# EPICS autosave request: iocBoot/ioc32IDMCTOptics/auto_settings.req
file "mctOptics.req", P=$(P), R=$(R)
file "mctOptics_settings.req", P=$(P), R=$(R)
